// TIA Portal V19 export
DATA_BLOCK "DB_Parameters"   // DB2
{ S7_Optimized_Access := 'TRUE'; DB_Accessible_From_OPC_UA := 'FALSE' }
// stored: DBAccessibleFromOPCUA false, DBAccessibleFromWebserver false, MemoryReserve 100
   VAR RETAIN
      CommMainPanel { ExternalAccessible := 'False'; ExternalVisible := 'False'; ExternalWritable := 'False'} : TCON_IP_v4;
      CommLeftRobot { ExternalAccessible := 'False'; ExternalVisible := 'False'; ExternalWritable := 'False'} : TCON_IP_v4;
      CommRightRobot { ExternalAccessible := 'False'; ExternalVisible := 'False'; ExternalWritable := 'False'} : TCON_IP_v4;
      tDelatBetweenReady { ExternalAccessible := 'False'; ExternalVisible := 'False'; ExternalWritable := 'False'} : Time := T#1s;
   END_VAR
BEGIN
   CommMainPanel.InterfaceId := 64;
   CommMainPanel.ID := 16#01;
   CommMainPanel.ConnectionType := 16#0B;
   CommMainPanel.ActiveEstablished := TRUE;
   CommMainPanel.RemoteAddress.ADDR[1] := 192;
   CommMainPanel.RemoteAddress.ADDR[2] := 168;
   CommMainPanel.RemoteAddress.ADDR[3] := 1;
   CommMainPanel.RemoteAddress.ADDR[4] := 20;
   CommMainPanel.RemotePort := 502;
   CommLeftRobot.InterfaceId := 64;
   CommLeftRobot.ID := 16#02;
   CommLeftRobot.ConnectionType := 16#0B;
   CommLeftRobot.ActiveEstablished := TRUE;
   CommLeftRobot.RemoteAddress.ADDR[1] := 192;
   CommLeftRobot.RemoteAddress.ADDR[2] := 168;
   CommLeftRobot.RemoteAddress.ADDR[3] := 1;
   CommLeftRobot.RemoteAddress.ADDR[4] := 21;
   CommLeftRobot.RemotePort := 502;
   CommRightRobot.InterfaceId := 64;
   CommRightRobot.ID := 16#03;
   CommRightRobot.ConnectionType := 16#0B;
   CommRightRobot.ActiveEstablished := TRUE;
   CommRightRobot.RemoteAddress.ADDR[1] := 192;
   CommRightRobot.RemoteAddress.ADDR[2] := 168;
   CommRightRobot.RemoteAddress.ADDR[3] := 1;
   CommRightRobot.RemoteAddress.ADDR[4] := 22;
   CommRightRobot.RemotePort := 503;
END_DATA_BLOCK
